INTERFACE I_AsyncResponseSessionData EXTENDS I_SessionData

METHOD PUBLIC Error
VAR_INPUT
	ErrorCode : T_MAXSTRING;
	Message : T_MAXSTRING;
END_VAR
END_METHOD

PROPERTY PUBLIC IsPending : BOOL
GET
END_GET
END_PROPERTY

METHOD PUBLIC Success
VAR_INPUT
END_VAR
END_METHOD

METHOD PUBLIC SuccessWithPayload
VAR_INPUT
	PayloadDataAddress : PVOID;
	PayloadDataSize : UDINT;
END_VAR
END_METHOD

PROPERTY PUBLIC SuggestedRetryDelayInMs : UDINT
GET
END_GET
SET
END_SET
END_PROPERTY

METHOD PUBLIC TryUpdateServerResponse : BOOL
VAR_INPUT
	Response : I_ServerResponse;
END_VAR
END_METHOD

END_INTERFACE

(* stored: Version 1.1.0.1, ProductVersion 3.1.4026.13
   Itf I_AsyncResponseSessionData: Id {37c0abde-ad3a-47ed-b6a1-b087262d1ff6}
   Method Error: Id {731f9662-674c-4231-bf68-63d33d8bc058}
   Property IsPending: Id {81bd7be5-52a3-455d-b074-542d0792efa3}
   Get Get: Id {34013b24-5966-4230-9ded-51629f26b3c3}
   Method Success: Id {e2870a85-528e-4ecc-98e5-a352304ff687}
   Method SuccessWithPayload: Id {907b657c-1f81-4409-aa60-e62e5c6d07a8}
   Property SuggestedRetryDelayInMs: Id {8d903687-92af-4eb9-aaea-69650571a103}
   Get Get: Id {93c0e8ea-6caa-4fe8-9550-8f43ed0f4993}
   Set Set: Id {fa81e1c6-cd39-42ce-b5b6-c99e9ca4d1f6}
   Method TryUpdateServerResponse: Id {22e85a6c-ee72-4365-9927-f5582d332d53} *)
